FUNCTION_BLOCK xPPUProduct IMPLEMENTS IProduct
VAR_INPUT
END_VAR
VAR_OUTPUT
END_VAR
VAR
	m_isPresent: BOOL;
	m_isLight: BOOL;
	m_isMetal: BOOL;
END_VAR

METHOD  Copy : BOOL
VAR_INPUT
	i_ptrOther: POINTER TO IProduct;
END_VAR
VAR
	m_ptrOther: POINTER TO xPPUProduct;
END_VAR
IF __QUERYPOINTER(i_ptrOther^, m_ptrOther) THEN
	m_isPresent := m_ptrOther^.IsPresent;
	m_isLight := m_ptrOther^.IsLight;
	m_isMetal := m_ptrOther^.IsMetal;
END_IF
END_METHOD

METHOD FB_init : BOOL
VAR_INPUT
	bInitRetains : BOOL; // if TRUE, the retain variables are initialized (warm start / cold start)
	bInCopyCode : BOOL;  // if TRUE, the instance afterwards gets moved into the copy code (online change)
END_VAR
END_METHOD

PROPERTY IsLight : BOOL
GET
IsLight := m_isLight;
END_GET
SET
m_isLight := IsLight;
END_SET
END_PROPERTY

PROPERTY IsMetal : BOOL
GET
IsMetal := m_isMetal;
END_GET
SET
m_isMetal := IsMetal;
END_SET
END_PROPERTY

PROPERTY IsPresent : BOOL
GET
IsPresent := m_isPresent;
END_GET
SET
m_isPresent := IsPresent;
END_SET
END_PROPERTY

PROPERTY Material : EProductTypes
GET
IF m_isPresent AND m_isLight AND NOT m_isMetal THEN
	Material := EProductTypes.white;
ELSIF m_isPresent AND NOT m_isLight AND NOT m_isMetal THEN
	Material := EProductTypes.black;
ELSIF m_isPresent AND m_isLight AND m_isMetal THEN
	Material := EProductTypes.metal;
ELSIF m_isPresent THEN
	Material := EProductTypes.unknown;
ELSE
	Material := EProductTypes.none;
END_IF
END_GET
END_PROPERTY

METHOD Reset : BOOL
m_isPresent := FALSE;
m_isLight := FALSE;
m_isMetal := FALSE;
END_METHOD

END_FUNCTION_BLOCK

(* stored: Version 1.1.0.1, ProductVersion 3.1.4024.9
   POU xPPUProduct: Id {91a53681-5c17-42d7-a486-9757a0df56c3}, SpecialFunc None
   Method Copy: Id {a392aebb-16ad-4571-b3a2-46e0c4375f0a}
   Method FB_init: Id {d8592a68-4c92-478b-a13b-d8564cba0d00}
   Property IsLight: Id {ea0efb76-d9ad-458d-8179-ec3b210fd4f5}
   Get Get: Id {715cfbdd-9448-4704-9468-e1e98c8fb22c}
   Set Set: Id {994323f3-e808-4b51-a892-9e65ddc3d29d}
   Property IsMetal: Id {92e12c06-9337-489e-8fd8-83f42c5d6469}
   Get Get: Id {638b79e7-ac93-42f8-baaf-393abe59adf5}
   Set Set: Id {e23154b7-63fc-445e-a847-97fbb8ca1b0f}
   Property IsPresent: Id {de916876-04ce-4f86-b84f-2e1990c87060}
   Get Get: Id {7512d3c5-a9f0-4cc2-83e7-95979571af3c}
   Set Set: Id {339221b5-e693-4097-ab00-7d3c50f91b00}
   Property Material: Id {dd1d66a9-edcd-4ad0-a48e-4d5be516b67d}
   Get Get: Id {613c400f-e2f1-4452-8c2b-37d9d64fd36c}
   Method Reset: Id {e588740d-ef36-4ed9-a03d-e9840f370d9a} *)
